TYPE ST_CoEIndSub :
STRUCT
    nIndex : WORD;
    nSubIndex : BYTE;
END_STRUCT
END_TYPE

(* stored: Version 1.1.0.1
   DUT ST_CoEIndSub: Id {62fd4c96-1a38-4aeb-82f8-1dcf9193e68a} *)
